TYPE E_SAFETY_GroupState :
(
	eSAFETY_GroupState_UNKNOWN		:= 0,
	eSAFETY_GroupState_RUN 			:= 1,
	eSAFETY_GroupState_STOP 		:= 2,
	eSAFETY_GroupState_SAFE			:= 3,
	eSAFETY_GroupState_ERROR		:= 4,
	eSAFETY_GroupState_RESET		:= 5
);
END_TYPE

(* stored: Version 1.1.0.1, ProductVersion 3.1.4022.12
   DUT E_SAFETY_GroupState: Id {b244b367-36df-428a-ab01-62748ebbee47} *)
